# B&R Automation Studio project MotionTestBenchMaster (part 30)

```iecst
                               VAR_RNS_SEQ.Mem.ContainersStop := TRUE;                                                 (* STEP: 51 *)
                               VAR_RNS_SEQ.Mem.ControlInsercion := FALSE;                                              (* STEP: 51 *)
                               VAR_RNS_SEQ.Mem.ControlContinous := FALSE;                                              (* STEP: 51 *)
                               VAR_RNS_SEQ.Mem.PBAbortEnable := FALSE;                                                 (* STEP: 51 PB Abort Sequence Enable*)
                               VAR_RNS_SEQ.Mem.PBStopEnable := TRUE;                                                   (* STEP: 51 PB Stop Sequence Enable*)
                               VAR_RNS_SEQ.Mem.PBStartEnable := FALSE;                                                 (* STEP: 51 PB Start Sequence Enable*)
                               VAR_RNS_SEQ.Mem.ByPassed := FALSE;                                                      (* STEP: 51 *)
                               VAR_RNS_SEQ.Mem.InsercionDevice := FALSE;                                               (* STEP: 51 *)
                               VAR_RNS_SEQ.Mem.AirTreatmentControl := FALSE;                                           (* STEP: 51 *)
                               VAR_RNS_SEQ.Mem.WaterTreatmentControl := FALSE;                                         (* STEP: 51 *)
                               VAR_RNS_SEQ.Mem.SpeedReductionControl := FALSE;                                         (* STEP: 51 *)
                               VAR_RNS_SEQ.Mem.ByPassRequest := FALSE;                                                 (* STEP: 51 *)
                               VAR_RNS_SEQ.Mem.CopAfterCipRequest := FALSE;                                            (* STEP: 51 *)
                               VAR_RNS_SEQ.Mem.NoBoNoSprayInsercion := FALSE;                                          (* STEP: 51 *)

                               VAR_RNS_SEQ.ITC.WTT_ProductRequest := FALSE;                                            (* STEP: 51 *)
                               VAR_RNS_SEQ.ITC.WTT_ProductionRunning := FALSE;                                         (* STEP: 51 *)

                       52..53: (* Spare Steps *)

                       54: (* DRAINING - Stopped *)

                               VAR_RNS_SEQ.Device.AVB224.AutoCnd := TRUE;                                              (* STEP: 54 AVB224*)
                               VAR_RNS_SEQ.Device.AVB224.EnableCnd := FALSE;
                               VAR_RNS_SEQ.Device.AVB228.AutoCnd := FALSE;                                             (* STEP: 54 AVB228*)
                               VAR_RNS_SEQ.Device.AVB228.EnableCnd := FALSE;
                               VAR_RNS_SEQ.Device.AVB234.AutoCnd := TRUE;                                              (* STEP: 54 AVB234*)
                               VAR_RNS_SEQ.Device.AVB234.EnableCnd := FALSE;
                               VAR_RNS_SEQ.Device.AVB261.AutoCnd := FALSE;                                             (* STEP: 54 AVB261*)
                               VAR_RNS_SEQ.Device.AVB261.EnableCnd := FALSE;
                               VAR_RNS_SEQ.Device.AVB264.AutoCnd := FALSE;                                             (* STEP: 54 AVB264*)
                               VAR_RNS_SEQ.Device.AVB264.EnableCnd := FALSE;
                               VAR_RNS_SEQ.Device.AVB265.AutoCnd := FALSE;                                             (* STEP: 54 AVB265*)
                               VAR_RNS_SEQ.Device.AVB265.EnableCnd := FALSE;
                               VAR_RNS_SEQ.Device.AVB266.AutoCnd := TRUE;                                              (* STEP: 54 AVB266*)
                               VAR_RNS_SEQ.Device.AVB266.EnableCnd := FALSE;
                               VAR_RNS_SEQ.Device.AVB267.AutoCnd := TRUE;                                              (* STEP: 54 AVB267*)
                               VAR_RNS_SEQ.Device.AVB267.EnableCnd := FALSE;
                               VAR_RNS_SEQ.Device.AVB268.AutoCnd := TRUE;                                              (* STEP: 54 AVB268*)
                               VAR_RNS_SEQ.Device.AVB268.EnableCnd := FALSE;
                               VAR_RNS_SEQ.Device.AVB273.AutoCnd := FALSE;                                             (* STEP: 54 AVB273*)
                               VAR_RNS_SEQ.Device.AVB273.EnableCnd := FALSE;
                               VAR_RNS_SEQ.Device.AVB294.AutoCnd := FALSE;                                             (* STEP: 54 AVB294*)
                               VAR_RNS_SEQ.Device.AVB294.EnableCnd := FALSE;

                               VAR_RNS_SEQ.Device.PPB209_PID.PID_Enable := FALSE;                                      (* STEP: 54 PPB209*)
                               VAR_RNS_SEQ.Device.PPB209_PID.PID_Mode := FALSE;
                               VAR_RNS_SEQ.Device.PPB209_PID.Auto_SP_Value := 0;
                               VAR_RNS_SEQ.Device.PPB209_PID.FIX_Value := 0;

                               VAR_RNS_SEQ.Device.RVB202_PID.PID_Enable := FALSE;                                      (* STEP: 54 *)
                               VAR_RNS_SEQ.Device.RVB202_PID.PID_Mode := FALSE;
                               VAR_RNS_SEQ.Device.RVB202_PID.Auto_SP_Value := 0;
                               VAR_RNS_SEQ.Device.RVB202_PID.FIX_Value := 0;

                               VAR_RNS_SEQ.Device.FSB220.ALR := FALSE;                                                 (* STEP: 54 FSB220*)
                               VAR_RNS_SEQ.Device.FSB220.WAIT_OFF := FALSE;
                               VAR_RNS_SEQ.Device.FSB220.WAIT_ON := FALSE;

                               VAR_RNS_SEQ.Device.LSB209.ALR := FALSE;                                                 (* STEP: 54 LSB209*)
                               VAR_RNS_SEQ.Device.LSB209.WAIT_OFF := FALSE;
                               VAR_RNS_SEQ.Device.LSB209.WAIT_ON := FALSE;

                               VAR_RNS_SEQ.Device.LSB210.ALR := FALSE;                                                 (* STEP: 54 LSB210*)
                               VAR_RNS_SEQ.Device.LSB210.WAIT_OFF := FALSE;
                               VAR_RNS_SEQ.Device.LSB210.WAIT_ON := FALSE;

                               VAR_RNS_SEQ.Device.LSB299.ALR := FALSE;                                                 (* STEP: 54 *)
                               VAR_RNS_SEQ.Device.LSB299.WAIT_OFF := FALSE;
                               VAR_RNS_SEQ.Device.LSB299.WAIT_ON := FALSE;

                               VAR_RNS_SEQ.Device.FSB201.ALR := FALSE;                                                 (* STEP: 54 FSB201*)
                               VAR_RNS_SEQ.Device.FSB201.WAIT_OFF := FALSE;
                               VAR_RNS_SEQ.Device.FSB201.WAIT_ON := FALSE;

                               VAR_RNS_SEQ.Device.FTB201.ALR_HighLimitEn := FALSE;                                     (* STEP: 54 FTB201*)
                               VAR_RNS_SEQ.Device.FTB201.ALR_HighLimitSP := 0;
                               VAR_RNS_SEQ.Device.FTB201.ALR_LowLimitEn := FALSE;
                               VAR_RNS_SEQ.Device.FTB201.ALR_LowLimitSP := 0;
                               VAR_RNS_SEQ.Device.FTB201.SP := 0;
                               VAR_RNS_SEQ.Device.FTB201.CMP := 0;
                               VAR_RNS_SEQ.Device.FTB201.MinDev := 0;
                               VAR_RNS_SEQ.Device.FTB201.MaxDev := 0;

                               VAR_RNS_SEQ.Device.FTB202.ALR_HighLimitEn := FALSE;                                     (* STEP: 54 FTB202*)
                               VAR_RNS_SEQ.Device.FTB202.ALR_HighLimitSP := 0;
                               VAR_RNS_SEQ.Device.FTB202.ALR_LowLimitEn := FALSE;
                               VAR_RNS_SEQ.Device.FTB202.ALR_LowLimitSP := 0;
                               VAR_RNS_SEQ.Device.FTB202.SP := 0;
                               VAR_RNS_SEQ.Device.FTB202.CMP := 0;
                               VAR_RNS_SEQ.Device.FTB202.MinDev := 0;
                               VAR_RNS_SEQ.Device.FTB202.MaxDev := 0;

                               VAR_RNS_SEQ.Device.PTB220.ALR_HighLimitEn := FALSE;                                     (* STEP: 54 PTB220*)
                               VAR_RNS_SEQ.Device.PTB220.ALR_HighLimitSP := 0;
                               VAR_RNS_SEQ.Device.PTB220.ALR_LowLimitEn := FALSE;
                               VAR_RNS_SEQ.Device.PTB220.ALR_LowLimitSP := 0;
                               VAR_RNS_SEQ.Device.PTB220.SP := 0;
                               VAR_RNS_SEQ.Device.PTB220.CMP := 0;
                               VAR_RNS_SEQ.Device.PTB220.MinDev := 0;
                               VAR_RNS_SEQ.Device.PTB220.MaxDev := 0;

                               VAR_RNS_SEQ.Device.PTB270.ALR_HighLimitEn := FALSE;                                     (* STEP: 54 PTB270*)
                               VAR_RNS_SEQ.Device.PTB270.ALR_HighLimitSP := 0;
                               VAR_RNS_SEQ.Device.PTB270.ALR_LowLimitEn := FALSE;
                               VAR_RNS_SEQ.Device.PTB270.ALR_LowLimitSP := 0;
                               VAR_RNS_SEQ.Device.PTB270.SP := 0;
                               VAR_RNS_SEQ.Device.PTB270.CMP := 0;
                               VAR_RNS_SEQ.Device.PTB270.MinDev := 0;
                               VAR_RNS_SEQ.Device.PTB270.MaxDev := 0;

                               VAR_RNS_SEQ.Device.LTB202.ALR_HighLimitEn := FALSE;                                     (* STEP: 54 LTB202*)
                               VAR_RNS_SEQ.Device.LTB202.ALR_HighLimitSP := 0;
                               VAR_RNS_SEQ.Device.LTB202.ALR_LowLimitEn := FALSE;
                               VAR_RNS_SEQ.Device.LTB202.ALR_LowLimitSP := 0;
                               VAR_RNS_SEQ.Device.LTB202.SP := 0;
                               VAR_RNS_SEQ.Device.LTB202.CMP := 0;
                               VAR_RNS_SEQ.Device.LTB202.MinDev := 0;
                               VAR_RNS_SEQ.Device.LTB202.MaxDev := 0;

                               VAR_RNS_SEQ.Device.PTB290.ALR_HighLimitEn := FALSE;                                     (* STEP: 54 PTB290*)
                               VAR_RNS_SEQ.Device.PTB290.ALR_HighLimitSP := 0;
                               VAR_RNS_SEQ.Device.PTB290.ALR_LowLimitEn := FALSE;
                               VAR_RNS_SEQ.Device.PTB290.ALR_LowLimitSP := 0;
                               VAR_RNS_SEQ.Device.PTB290.SP := 0;
                               VAR_RNS_SEQ.Device.PTB290.CMP := 0;
                               VAR_RNS_SEQ.Device.PTB290.MinDev := 0;
                               VAR_RNS_SEQ.Device.PTB290.MaxDev := 0;

                               VAR_RNS_SEQ.Mem.ContainersStop := TRUE;                                                 (* STEP: 54 *)
                               VAR_RNS_SEQ.Mem.ControlInsercion := FALSE;                                              (* STEP: 54 *)
                               VAR_RNS_SEQ.Mem.ControlContinous := FALSE;                                              (* STEP: 54 *)
                               VAR_RNS_SEQ.Mem.PBAbortEnable := FALSE;                                                 (* STEP: 54 PB Abort Sequence Enable*)
                               VAR_RNS_SEQ.Mem.PBStopEnable := TRUE;                                                   (* STEP: 54 PB Stop Sequence Enable*)
                               VAR_RNS_SEQ.Mem.PBStartEnable := FALSE;                                                 (* STEP: 54 PB Start Sequence Enable*)
                               VAR_RNS_SEQ.Mem.ByPassed := FALSE;                                                      (* STEP: 54 *)
                               VAR_RNS_SEQ.Mem.InsercionDevice := FALSE;                                               (* STEP: 54 *)
                               VAR_RNS_SEQ.Mem.AirTreatmentControl := FALSE;                                           (* STEP: 54 *)
                               VAR_RNS_SEQ.Mem.WaterTreatmentControl := FALSE;                                         (* STEP: 54 *)
                               VAR_RNS_SEQ.Mem.SpeedReductionControl := FALSE;                                         (* STEP: 54 *)
                               VAR_RNS_SEQ.Mem.ByPassRequest := FALSE;                                                 (* STEP: 54 *)
                               VAR_RNS_SEQ.Mem.CopAfterCipRequest := FALSE;                                            (* STEP: 54 *)
                               VAR_RNS_SEQ.Mem.NoBoNoSprayInsercion := FALSE;                                          (* STEP: 54 *)

                               VAR_RNS_SEQ.ITC.WTT_ProductRequest := FALSE;                                            (* STEP: 54 *)
                               VAR_RNS_SEQ.ITC.WTT_ProductionRunning := FALSE;                                         (* STEP: 54 *)

                       55: (* DRAINING - Circuit emptying during COP *)

                               VAR_RNS_SEQ.Device.AVB224.AutoCnd := FALSE;                                             (* STEP: 55 AVB224*)
                               VAR_RNS_SEQ.Device.AVB224.EnableCnd := FALSE;
                               VAR_RNS_SEQ.Device.AVB228.AutoCnd := FALSE;                                             (* STEP: 55 AVB228*)
                               VAR_RNS_SEQ.Device.AVB228.EnableCnd := FALSE;
                               VAR_RNS_SEQ.Device.AVB234.AutoCnd := FALSE;                                             (* STEP: 55 AVB234*)
                               VAR_RNS_SEQ.Device.AVB234.EnableCnd := FALSE;
                               VAR_RNS_SEQ.Device.AVB261.AutoCnd := FALSE;                                             (* STEP: 55 AVB261*)
                               VAR_RNS_SEQ.Device.AVB261.EnableCnd := FALSE;
                               VAR_RNS_SEQ.Device.AVB264.AutoCnd := FALSE;                                             (* STEP: 55 AVB264*)
                               VAR_RNS_SEQ.Device.AVB264.EnableCnd := FALSE;
                               VAR_RNS_SEQ.Device.AVB265.AutoCnd := FALSE;                                             (* STEP: 55 AVB265*)
                               VAR_RNS_SEQ.Device.AVB265.EnableCnd := FALSE;
                               VAR_RNS_SEQ.Device.AVB266.AutoCnd := FALSE;                                             (* STEP: 55 AVB266*)
                               VAR_RNS_SEQ.Device.AVB266.EnableCnd := FALSE;
                               VAR_RNS_SEQ.Device.AVB267.AutoCnd := FALSE;                                             (* STEP: 55 AVB267*)
                               VAR_RNS_SEQ.Device.AVB267.EnableCnd := FALSE;
                               VAR_RNS_SEQ.Device.AVB268.AutoCnd := TRUE;                                              (* STEP: 55 AVB268*)
                               VAR_RNS_SEQ.Device.AVB268.EnableCnd := FALSE;
                               VAR_RNS_SEQ.Device.AVB273.AutoCnd := FALSE;                                             (* STEP: 55 AVB273*)
                               VAR_RNS_SEQ.Device.AVB273.EnableCnd := FALSE;
                               VAR_RNS_SEQ.Device.AVB294.AutoCnd := FALSE;                                             (* STEP: 55 AVB294*)
                               VAR_RNS_SEQ.Device.AVB294.EnableCnd := FALSE;

                               VAR_RNS_SEQ.Device.PPB209_PID.PID_Enable := FALSE;                                      (* STEP: 55 PPB209*)
                               VAR_RNS_SEQ.Device.PPB209_PID.PID_Mode := FALSE;
                               VAR_RNS_SEQ.Device.PPB209_PID.Auto_SP_Value := 0;
                               VAR_RNS_SEQ.Device.PPB209_PID.FIX_Value := 0;

                               VAR_RNS_SEQ.Device.RVB202_PID.PID_Enable := FALSE;                                      (* STEP: 55 *)
                               VAR_RNS_SEQ.Device.RVB202_PID.PID_Mode := FALSE;
                               VAR_RNS_SEQ.Device.RVB202_PID.Auto_SP_Value := 0;
                               VAR_RNS_SEQ.Device.RVB202_PID.FIX_Value := 0;

                               VAR_RNS_SEQ.Device.FSB220.ALR := FALSE;                                                 (* STEP: 55 FSB220*)
                               VAR_RNS_SEQ.Device.FSB220.WAIT_OFF := FALSE;
                               VAR_RNS_SEQ.Device.FSB220.WAIT_ON := FALSE;

                               VAR_RNS_SEQ.Device.LSB209.ALR := FALSE;                                                 (* STEP: 55 LSB209*)
                               VAR_RNS_SEQ.Device.LSB209.WAIT_OFF := FALSE;
                               VAR_RNS_SEQ.Device.LSB209.WAIT_ON := FALSE;

                               VAR_RNS_SEQ.Device.LSB210.ALR := FALSE;                                                 (* STEP: 55 LSB210*)
                               VAR_RNS_SEQ.Device.LSB210.WAIT_OFF := FALSE;
                               VAR_RNS_SEQ.Device.LSB210.WAIT_ON := FALSE;

                               VAR_RNS_SEQ.Device.LSB299.ALR := FALSE;                                                 (* STEP: 55 *)
                               VAR_RNS_SEQ.Device.LSB299.WAIT_OFF := FALSE;
                               VAR_RNS_SEQ.Device.LSB299.WAIT_ON := FALSE;

                               VAR_RNS_SEQ.Device.FSB201.ALR := FALSE;                                                 (* STEP: 55 FSB201*)
                               VAR_RNS_SEQ.Device.FSB201.WAIT_OFF := FALSE;
                               VAR_RNS_SEQ.Device.FSB201.WAIT_ON := FALSE;

                               VAR_RNS_SEQ.Device.FTB201.ALR_HighLimitEn := FALSE;                                     (* STEP: 55 FTB201*)
                               VAR_RNS_SEQ.Device.FTB201.ALR_HighLimitSP := 0;
                               VAR_RNS_SEQ.Device.FTB201.ALR_LowLimitEn := FALSE;
                               VAR_RNS_SEQ.Device.FTB201.ALR_LowLimitSP := 0;
                               VAR_RNS_SEQ.Device.FTB201.SP := 0;
                               VAR_RNS_SEQ.Device.FTB201.CMP := 0;
                               VAR_RNS_SEQ.Device.FTB201.MinDev := 0;
                               VAR_RNS_SEQ.Device.FTB201.MaxDev := 0;

                               VAR_RNS_SEQ.Device.FTB202.ALR_HighLimitEn := FALSE;                                     (* STEP: 55 FTB202*)
                               VAR_RNS_SEQ.Device.FTB202.ALR_HighLimitSP := 0;
                               VAR_RNS_SEQ.Device.FTB202.ALR_LowLimitEn := FALSE;
                               VAR_RNS_SEQ.Device.FTB202.ALR_LowLimitSP := 0;
                               VAR_RNS_SEQ.Device.FTB202.SP := 0;
                               VAR_RNS_SEQ.Device.FTB202.CMP := 0;
                               VAR_RNS_SEQ.Device.FTB202.MinDev := 0;
                               VAR_RNS_SEQ.Device.FTB202.MaxDev := 0;

                               VAR_RNS_SEQ.Device.PTB220.ALR_HighLimitEn := FALSE;                                     (* STEP: 55 PTB220*)
                               VAR_RNS_SEQ.Device.PTB220.ALR_HighLimitSP := 0;
                               VAR_RNS_SEQ.Device.PTB220.ALR_LowLimitEn := FALSE;
                               VAR_RNS_SEQ.Device.PTB220.ALR_LowLimitSP := 0;
                               VAR_RNS_SEQ.Device.PTB220.SP := 0;
                               VAR_RNS_SEQ.Device.PTB220.CMP := 0;
                               VAR_RNS_SEQ.Device.PTB220.MinDev := 0;
                               VAR_RNS_SEQ.Device.PTB220.MaxDev := 0;

                               VAR_RNS_SEQ.Device.PTB270.ALR_HighLimitEn := FALSE;                                     (* STEP: 55 PTB270*)
                               VAR_RNS_SEQ.Device.PTB270.ALR_HighLimitSP := 0;
                               VAR_RNS_SEQ.Device.PTB270.ALR_LowLimitEn := FALSE;
                               VAR_RNS_SEQ.Device.PTB270.ALR_LowLimitSP := 0;
                               VAR_RNS_SEQ.Device.PTB270.SP := 0;
                               VAR_RNS_SEQ.Device.PTB270.CMP := 0;
                               VAR_RNS_SEQ.Device.PTB270.MinDev := 0;
                               VAR_RNS_SEQ.Device.PTB270.MaxDev := 0;

                               VAR_RNS_SEQ.Device.LTB202.ALR_HighLimitEn := FALSE;                                     (* STEP: 55 LTB202*)
                               VAR_RNS_SEQ.Device.LTB202.ALR_HighLimitSP := 0;
                               VAR_RNS_SEQ.Device.LTB202.ALR_LowLimitEn := FALSE;
                               VAR_RNS_SEQ.Device.LTB202.ALR_LowLimitSP := 0;
                               VAR_RNS_SEQ.Device.LTB202.SP := 0;
                               VAR_RNS_SEQ.Device.LTB202.CMP := 0;
                               VAR_RNS_SEQ.Device.LTB202.MinDev := 0;
                               VAR_RNS_SEQ.Device.LTB202.MaxDev := 0;

                               VAR_RNS_SEQ.Device.PTB290.ALR_HighLimitEn := FALSE;                                     (* STEP: 55 PTB290*)
                               VAR_RNS_SEQ.Device.PTB290.ALR_HighLimitSP := 0;
                               VAR_RNS_SEQ.Device.PTB290.ALR_LowLimitEn := FALSE;
                               VAR_RNS_SEQ.Device.PTB290.ALR_LowLimitSP := 0;
                               VAR_RNS_SEQ.Device.PTB290.SP := 0;
                               VAR_RNS_SEQ.Device.PTB290.CMP := 0;
                               VAR_RNS_SEQ.Device.PTB290.MinDev := 0;
                               VAR_RNS_SEQ.Device.PTB290.MaxDev := 0;

                               VAR_RNS_SEQ.Mem.ContainersStop := TRUE;                                                 (* STEP: 55 *)
                               VAR_RNS_SEQ.Mem.ControlInsercion := FALSE;                                              (* STEP: 55 *)
                               VAR_RNS_SEQ.Mem.ControlContinous := FALSE;                                              (* STEP: 55 *)
                               VAR_RNS_SEQ.Mem.PBAbortEnable := FALSE;                                                 (* STEP: 55 PB Abort Sequence Enable*)
                               VAR_RNS_SEQ.Mem.PBStopEnable := FALSE;                                                  (* STEP: 55 PB Stop Sequence Enable*)
                               VAR_RNS_SEQ.Mem.PBStartEnable := FALSE;                                                 (* STEP: 55 PB Start Sequence Enable*)
                               VAR_RNS_SEQ.Mem.ByPassed := FALSE;                                                      (* STEP: 55 *)
                               VAR_RNS_SEQ.Mem.InsercionDevice := FALSE;                                               (* STEP: 55 *)
                               VAR_RNS_SEQ.Mem.AirTreatmentControl := FALSE;                                           (* STEP: 55 *)
                               VAR_RNS_SEQ.Mem.WaterTreatmentControl := FALSE;                                         (* STEP: 55 *)
                               VAR_RNS_SEQ.Mem.SpeedReductionControl := TRUE;                                          (* STEP: 55 *)
                               VAR_RNS_SEQ.Mem.ByPassRequest := FALSE;                                                 (* STEP: 55 *)
                               VAR_RNS_SEQ.Mem.CopAfterCipRequest := TRUE;                                             (* STEP: 55 *)
                               VAR_RNS_SEQ.Mem.NoBoNoSprayInsercion := FALSE;                                          (* STEP: 55 *)

                               VAR_RNS_SEQ.ITC.WTT_ProductRequest := FALSE;                                            (* STEP: 55 *)
                               VAR_RNS_SEQ.ITC.WTT_ProductionRunning := FALSE;                                         (* STEP: 55 *)

                       56..69: (* Spare Steps *)

                       70: (* CONTROL - Check Selection and Speed *)

                               VAR_RNS_SEQ.Device.AVB224.AutoCnd := FALSE;                                             (* STEP: 70 AVB224*)
                               VAR_RNS_SEQ.Device.AVB224.EnableCnd := FALSE;
                               VAR_RNS_SEQ.Device.AVB228.AutoCnd := FALSE;                                             (* STEP: 70 AVB228*)
                               VAR_RNS_SEQ.Device.AVB228.EnableCnd := FALSE;
                               VAR_RNS_SEQ.Device.AVB234.AutoCnd := FALSE;                                             (* STEP: 70 AVB234*)
                               VAR_RNS_SEQ.Device.AVB234.EnableCnd := FALSE;
                               VAR_RNS_SEQ.Device.AVB261.AutoCnd := FALSE;                                             (* STEP: 70 AVB261*)
                               VAR_RNS_SEQ.Device.AVB261.EnableCnd := FALSE;
                               VAR_RNS_SEQ.Device.AVB264.AutoCnd := FALSE;                                             (* STEP: 70 AVB264*)
                               VAR_RNS_SEQ.Device.AVB264.EnableCnd := FALSE;
                               VAR_RNS_SEQ.Device.AVB265.AutoCnd := FALSE;                                             (* STEP: 70 AVB265*)
                               VAR_RNS_SEQ.Device.AVB265.EnableCnd := FALSE;
                               VAR_RNS_SEQ.Device.AVB266.AutoCnd := FALSE;                                             (* STEP: 70 AVB266*)
                               VAR_RNS_SEQ.Device.AVB266.EnableCnd := FALSE;
                               VAR_RNS_SEQ.Device.AVB267.AutoCnd := FALSE;                                             (* STEP: 70 AVB267*)
                               VAR_RNS_SEQ.Device.AVB267.EnableCnd := FALSE;
                               VAR_RNS_SEQ.Device.AVB268.AutoCnd := FALSE;                                             (* STEP: 70 AVB268*)
                               VAR_RNS_SEQ.Device.AVB268.EnableCnd := FALSE;
                               VAR_RNS_SEQ.Device.AVB273.AutoCnd := FALSE;                                             (* STEP: 70 AVB273*)
                               VAR_RNS_SEQ.Device.AVB273.EnableCnd := FALSE;
                               VAR_RNS_SEQ.Device.AVB294.AutoCnd := FALSE;                                             (* STEP: 70 AVB294*)
                               VAR_RNS_SEQ.Device.AVB294.EnableCnd := FALSE;

                               VAR_RNS_SEQ.Device.PPB209_PID.PID_Enable := FALSE;                                      (* STEP: 70 PPB209*)
                               VAR_RNS_SEQ.Device.PPB209_PID.PID_Mode := FALSE;
                               VAR_RNS_SEQ.Device.PPB209_PID.Auto_SP_Value := 0;
                               VAR_RNS_SEQ.Device.PPB209_PID.FIX_Value := 0;

                               VAR_RNS_SEQ.Device.RVB202_PID.PID_Enable := FALSE;                                      (* STEP: 70 *)
                               VAR_RNS_SEQ.Device.RVB202_PID.PID_Mode := FALSE;
                               VAR_RNS_SEQ.Device.RVB202_PID.Auto_SP_Value := 0;
                               VAR_RNS_SEQ.Device.RVB202_PID.FIX_Value := 0;

                               VAR_RNS_SEQ.Device.FSB220.ALR := FALSE;                                                 (* STEP: 70 FSB220*)
                               VAR_RNS_SEQ.Device.FSB220.WAIT_OFF := FALSE;
                               VAR_RNS_SEQ.Device.FSB220.WAIT_ON := FALSE;

                               VAR_RNS_SEQ.Device.LSB209.ALR := FALSE;                                                 (* STEP: 70 LSB209*)
                               VAR_RNS_SEQ.Device.LSB209.WAIT_OFF := FALSE;
                               VAR_RNS_SEQ.Device.LSB209.WAIT_ON := FALSE;

                               VAR_RNS_SEQ.Device.LSB210.ALR := FALSE;                                                 (* STEP: 70 LSB210*)
                               VAR_RNS_SEQ.Device.LSB210.WAIT_OFF := FALSE;
                               VAR_RNS_SEQ.Device.LSB210.WAIT_ON := FALSE;

                               VAR_RNS_SEQ.Device.LSB299.ALR := FALSE;                                                 (* STEP: 70 *)
                               VAR_RNS_SEQ.Device.LSB299.WAIT_OFF := FALSE;
                               VAR_RNS_SEQ.Device.LSB299.WAIT_ON := FALSE;

                               VAR_RNS_SEQ.Device.FSB201.ALR := FALSE;                                                 (* STEP: 70 FSB201*)
                               VAR_RNS_SEQ.Device.FSB201.WAIT_OFF := FALSE;
                               VAR_RNS_SEQ.Device.FSB201.WAIT_ON := FALSE;

                               VAR_RNS_SEQ.Device.FTB201.ALR_HighLimitEn := FALSE;                                     (* STEP: 70 FTB201*)
                               VAR_RNS_SEQ.Device.FTB201.ALR_HighLimitSP := 0;
                               VAR_RNS_SEQ.Device.FTB201.ALR_LowLimitEn := FALSE;
                               VAR_RNS_SEQ.Device.FTB201.ALR_LowLimitSP := 0;
                               VAR_RNS_SEQ.Device.FTB201.SP := 0;
                               VAR_RNS_SEQ.Device.FTB201.CMP := 0;
                               VAR_RNS_SEQ.Device.FTB201.MinDev := 0;
                               VAR_RNS_SEQ.Device.FTB201.MaxDev := 0;

                               VAR_RNS_SEQ.Device.FTB202.ALR_HighLimitEn := FALSE;                                     (* STEP: 70 FTB202*)
                               VAR_RNS_SEQ.Device.FTB202.ALR_HighLimitSP := 0;
                               VAR_RNS_SEQ.Device.FTB202.ALR_LowLimitEn := FALSE;
                               VAR_RNS_SEQ.Device.FTB202.ALR_LowLimitSP := 0;
                               VAR_RNS_SEQ.Device.FTB202.SP := 0;
                               VAR_RNS_SEQ.Device.FTB202.CMP := 0;
                               VAR_RNS_SEQ.Device.FTB202.MinDev := 0;
                               VAR_RNS_SEQ.Device.FTB202.MaxDev := 0;

                               VAR_RNS_SEQ.Device.PTB220.ALR_HighLimitEn := FALSE;                                     (* STEP: 70 PTB220*)
                               VAR_RNS_SEQ.Device.PTB220.ALR_HighLimitSP := 0;
                               VAR_RNS_SEQ.Device.PTB220.ALR_LowLimitEn := FALSE;
                               VAR_RNS_SEQ.Device.PTB220.ALR_LowLimitSP := 0;
                               VAR_RNS_SEQ.Device.PTB220.SP := 0;
                               VAR_RNS_SEQ.Device.PTB220.CMP := 0;
                               VAR_RNS_SEQ.Device.PTB220.MinDev := 0;
                               VAR_RNS_SEQ.Device.PTB220.MaxDev := 0;

                               VAR_RNS_SEQ.Device.PTB270.ALR_HighLimitEn := FALSE;                                     (* STEP: 70 PTB270*)
                               VAR_RNS_SEQ.Device.PTB270.ALR_HighLimitSP := 0;
                               VAR_RNS_SEQ.Device.PTB270.ALR_LowLimitEn := FALSE;
                               VAR_RNS_SEQ.Device.PTB270.ALR_LowLimitSP := 0;
                               VAR_RNS_SEQ.Device.PTB270.SP := 0;
                               VAR_RNS_SEQ.Device.PTB270.CMP := 0;
                               VAR_RNS_SEQ.Device.PTB270.MinDev := 0;
                               VAR_RNS_SEQ.Device.PTB270.MaxDev := 0;

                               VAR_RNS_SEQ.Device.LTB202.ALR_HighLimitEn := FALSE;                                     (* STEP: 70 LTB202*)
                               VAR_RNS_SEQ.Device.LTB202.ALR_HighLimitSP := 0;
                               VAR_RNS_SEQ.Device.LTB202.ALR_LowLimitEn := FALSE;
                               VAR_RNS_SEQ.Device.LTB202.ALR_LowLimitSP := 0;
                               VAR_RNS_SEQ.Device.LTB202.SP := 0;
                               VAR_RNS_SEQ.Device.LTB202.CMP := 0;
                               VAR_RNS_SEQ.Device.LTB202.MinDev := 0;
                               VAR_RNS_SEQ.Device.LTB202.MaxDev := 0;

                               VAR_RNS_SEQ.Device.PTB290.ALR_HighLimitEn := FALSE;                                     (* STEP: 70 PTB290*)
                               VAR_RNS_SEQ.Device.PTB290.ALR_HighLimitSP := 0;
                               VAR_RNS_SEQ.Device.PTB290.ALR_LowLimitEn := FALSE;
                               VAR_RNS_SEQ.Device.PTB290.ALR_LowLimitSP := 0;
                               VAR_RNS_SEQ.Device.PTB290.SP := 0;
                               VAR_RNS_SEQ.Device.PTB290.CMP := 0;
                               VAR_RNS_SEQ.Device.PTB290.MinDev := 0;
                               VAR_RNS_SEQ.Device.PTB290.MaxDev := 0;

                               VAR_RNS_SEQ.Mem.ContainersStop := TRUE;                                                 (* STEP: 70 *)
                               VAR_RNS_SEQ.Mem.ControlInsercion := FALSE;                                              (* STEP: 70 *)
                               VAR_RNS_SEQ.Mem.ControlContinous := FALSE;                                              (* STEP: 70 *)
                               VAR_RNS_SEQ.Mem.PBAbortEnable := TRUE;                                                  (* STEP: 70 PB Abort Sequence Enable*)
                               VAR_RNS_SEQ.Mem.PBStopEnable := TRUE;                                                   (* STEP: 70 PB Stop Sequence Enable*)
                               VAR_RNS_SEQ.Mem.PBStartEnable := FALSE;                                                 (* STEP: 70 PB Start Sequence Enable*)
                               VAR_RNS_SEQ.Mem.ByPassed := FALSE;                                                      (* STEP: 70 *)
                               VAR_RNS_SEQ.Mem.InsercionDevice := FALSE;                                               (* STEP: 70 *)
                               VAR_RNS_SEQ.Mem.AirTreatmentControl := FALSE;                                           (* STEP: 70 *)
                               VAR_RNS_SEQ.Mem.WaterTreatmentControl := FALSE;                                         (* STEP: 70 *)
                               VAR_RNS_SEQ.Mem.SpeedReductionControl := TRUE;                                          (* STEP: 70 *)
                               VAR_RNS_SEQ.Mem.ByPassRequest := FALSE;                                                 (* STEP: 70 *)
                               VAR_RNS_SEQ.Mem.CopAfterCipRequest := FALSE;                                            (* STEP: 70 *)
                               VAR_RNS_SEQ.Mem.NoBoNoSprayInsercion := FALSE;                                          (* STEP: 70 *)

                               VAR_RNS_SEQ.ITC.WTT_ProductRequest := FALSE;                                            (* STEP: 70 *)
                               VAR_RNS_SEQ.ITC.WTT_ProductionRunning := FALSE;                                         (* STEP: 70 *)

                       71: (* CONTROL - Insercion Device *)

                               VAR_RNS_SEQ.Device.AVB224.AutoCnd := FALSE;                                             (* STEP: 71 AVB224*)
                               VAR_RNS_SEQ.Device.AVB224.EnableCnd := FALSE;
                               VAR_RNS_SEQ.Device.AVB228.AutoCnd := TRUE;                                              (* STEP: 71 AVB228*)
                               VAR_RNS_SEQ.Device.AVB228.EnableCnd := FALSE;
                               VAR_RNS_SEQ.Device.AVB234.AutoCnd := FALSE;                                             (* STEP: 71 AVB234*)
                               VAR_RNS_SEQ.Device.AVB234.EnableCnd := FALSE;
                               VAR_RNS_SEQ.Device.AVB261.AutoCnd := TRUE;                                              (* STEP: 71 AVB261*)
                               VAR_RNS_SEQ.Device.AVB261.EnableCnd := FALSE;
                               VAR_RNS_SEQ.Device.AVB264.AutoCnd := FALSE;                                             (* STEP: 71 AVB264*)
                               VAR_RNS_SEQ.Device.AVB264.EnableCnd := FALSE;
                               VAR_RNS_SEQ.Device.AVB265.AutoCnd := FALSE;                                             (* STEP: 71 AVB265*)
                               VAR_RNS_SEQ.Device.AVB265.EnableCnd := FALSE;
                               VAR_RNS_SEQ.Device.AVB266.AutoCnd := FALSE;                                             (* STEP: 71 AVB266*)
                               VAR_RNS_SEQ.Device.AVB266.EnableCnd := FALSE;
                               VAR_RNS_SEQ.Device.AVB267.AutoCnd := FALSE;                                             (* STEP: 71 AVB267*)
                               VAR_RNS_SEQ.Device.AVB267.EnableCnd := FALSE;
                               VAR_RNS_SEQ.Device.AVB268.AutoCnd := FALSE;                                             (* STEP: 71 AVB268*)
                               VAR_RNS_SEQ.Device.AVB268.EnableCnd := FALSE;
                               VAR_RNS_SEQ.Device.AVB273.AutoCnd := FALSE;                                             (* STEP: 71 AVB273*)
                               VAR_RNS_SEQ.Device.AVB273.EnableCnd := FALSE;
                               VAR_RNS_SEQ.Device.AVB294.AutoCnd := FALSE;                                             (* STEP: 71 AVB294*)
                               VAR_RNS_SEQ.Device.AVB294.EnableCnd := FALSE;

                               VAR_RNS_SEQ.Device.PPB209_PID.PID_Enable := FALSE;                                      (* STEP: 71 PPB209*)
                               VAR_RNS_SEQ.Device.PPB209_PID.PID_Mode := FALSE;
                               VAR_RNS_SEQ.Device.PPB209_PID.Auto_SP_Value := 0;
                               VAR_RNS_SEQ.Device.PPB209_PID.FIX_Value := 0;

                               VAR_RNS_SEQ.Device.RVB202_PID.PID_Enable := FALSE;                                      (* STEP: 71 *)
                               VAR_RNS_SEQ.Device.RVB202_PID.PID_Mode := FALSE;
                               VAR_RNS_SEQ.Device.RVB202_PID.Auto_SP_Value := 0;
                               VAR_RNS_SEQ.Device.RVB202_PID.FIX_Value := 0;

                               VAR_RNS_SEQ.Device.FSB220.ALR := TRUE;                                                  (* STEP: 71 FSB220*)
                               VAR_RNS_SEQ.Device.FSB220.WAIT_OFF := FALSE;
                               VAR_RNS_SEQ.Device.FSB220.WAIT_ON := TRUE;

                               VAR_RNS_SEQ.Device.LSB209.ALR := FALSE;                                                 (* STEP: 71 LSB209*)
                               VAR_RNS_SEQ.Device.LSB209.WAIT_OFF := FALSE;
                               VAR_RNS_SEQ.Device.LSB209.WAIT_ON := FALSE;

                               VAR_RNS_SEQ.Device.LSB210.ALR := FALSE;                                                 (* STEP: 71 LSB210*)
                               VAR_RNS_SEQ.Device.LSB210.WAIT_OFF := FALSE;
                               VAR_RNS_SEQ.Device.LSB210.WAIT_ON := FALSE;

                               VAR_RNS_SEQ.Device.LSB299.ALR := FALSE;                                                 (* STEP: 71 *)
                               VAR_RNS_SEQ.Device.LSB299.WAIT_OFF := FALSE;
                               VAR_RNS_SEQ.Device.LSB299.WAIT_ON := FALSE;

                               VAR_RNS_SEQ.Device.FSB201.ALR := TRUE;                                                  (* STEP: 71 FSB201*)
                               VAR_RNS_SEQ.Device.FSB201.WAIT_OFF := FALSE;
                               VAR_RNS_SEQ.Device.FSB201.WAIT_ON := TRUE;

                               VAR_RNS_SEQ.Device.FTB201.ALR_HighLimitEn := FALSE;                                     (* STEP: 71 FTB201*)
                               VAR_RNS_SEQ.Device.FTB201.ALR_HighLimitSP := 0;
                               VAR_RNS_SEQ.Device.FTB201.ALR_LowLimitEn := FALSE;
                               VAR_RNS_SEQ.Device.FTB201.ALR_LowLimitSP := 0;
                               VAR_RNS_SEQ.Device.FTB201.SP := 0;
                               VAR_RNS_SEQ.Device.FTB201.CMP := 0;
                               VAR_RNS_SEQ.Device.FTB201.MinDev := 0;
                               VAR_RNS_SEQ.Device.FTB201.MaxDev := 0;

                               VAR_RNS_SEQ.Device.FTB202.ALR_HighLimitEn := FALSE;                                     (* STEP: 71 FTB202*)
                               VAR_RNS_SEQ.Device.FTB202.ALR_HighLimitSP := 0;
                               VAR_RNS_SEQ.Device.FTB202.ALR_LowLimitEn := FALSE;
                               VAR_RNS_SEQ.Device.FTB202.ALR_LowLimitSP := 0;
                               VAR_RNS_SEQ.Device.FTB202.SP := 0;
                               VAR_RNS_SEQ.Device.FTB202.CMP := 0;
                               VAR_RNS_SEQ.Device.FTB202.MinDev := 0;
                               VAR_RNS_SEQ.Device.FTB202.MaxDev := 0;

                               VAR_RNS_SEQ.Device.PTB220.ALR_HighLimitEn := FALSE;                                     (* STEP: 71 PTB220*)
                               VAR_RNS_SEQ.Device.PTB220.ALR_HighLimitSP := 0;
                               VAR_RNS_SEQ.Device.PTB220.ALR_LowLimitEn := FALSE;
                               VAR_RNS_SEQ.Device.PTB220.ALR_LowLimitSP := 0;
                               VAR_RNS_SEQ.Device.PTB220.SP := 0;
                               VAR_RNS_SEQ.Device.PTB220.CMP := 0;
                               VAR_RNS_SEQ.Device.PTB220.MinDev := 0;
                               VAR_RNS_SEQ.Device.PTB220.MaxDev := 0;

                               VAR_RNS_SEQ.Device.PTB270.ALR_HighLimitEn := FALSE;                                     (* STEP: 71 PTB270*)
                               VAR_RNS_SEQ.Device.PTB270.ALR_HighLimitSP := 0;
                               VAR_RNS_SEQ.Device.PTB270.ALR_LowLimitEn := FALSE;
                               VAR_RNS_SEQ.Device.PTB270.ALR_LowLimitSP := 0;
                               VAR_RNS_SEQ.Device.PTB270.SP := 0;
                               VAR_RNS_SEQ.Device.PTB270.CMP := 0;
                               VAR_RNS_SEQ.Device.PTB270.MinDev := 0;
                               VAR_RNS_SEQ.Device.PTB270.MaxDev := 0;

                               VAR_RNS_SEQ.Device.LTB202.ALR_HighLimitEn := FALSE;                                     (* STEP: 71 LTB202*)
                               VAR_RNS_SEQ.Device.LTB202.ALR_HighLimitSP := 0;
                               VAR_RNS_SEQ.Device.LTB202.ALR_LowLimitEn := FALSE;
                               VAR_RNS_SEQ.Device.LTB202.ALR_LowLimitSP := 0;
                               VAR_RNS_SEQ.Device.LTB202.SP := 0;
                               VAR_RNS_SEQ.Device.LTB202.CMP := 0;
                               VAR_RNS_SEQ.Device.LTB202.MinDev := 0;
                               VAR_RNS_SEQ.Device.LTB202.MaxDev := 0;

                               VAR_RNS_SEQ.Device.PTB290.ALR_HighLimitEn := FALSE;                                     (* STEP: 71 PTB290*)
                               VAR_RNS_SEQ.Device.PTB290.ALR_HighLimitSP := 0;
                               VAR_RNS_SEQ.Device.PTB290.ALR_LowLimitEn := FALSE;
                               VAR_RNS_SEQ.Device.PTB290.ALR_LowLimitSP := 0;
                               VAR_RNS_SEQ.Device.PTB290.SP := 0;
                               VAR_RNS_SEQ.Device.PTB290.CMP := 0;
                               VAR_RNS_SEQ.Device.PTB290.MinDev := 0;
                               VAR_RNS_SEQ.Device.PTB290.MaxDev := 0;

                               VAR_RNS_SEQ.Mem.ContainersStop := TRUE;                                                 (* STEP: 71 *)
                               VAR_RNS_SEQ.Mem.ControlInsercion := FALSE;                                              (* STEP: 71 *)
                               VAR_RNS_SEQ.Mem.ControlContinous := FALSE;                                              (* STEP: 71 *)
                               VAR_RNS_SEQ.Mem.PBAbortEnable := TRUE;                                                  (* STEP: 71 PB Abort Sequence Enable*)
                               VAR_RNS_SEQ.Mem.PBStopEnable := TRUE;                                                   (* STEP: 71 PB Stop Sequence Enable*)
                               VAR_RNS_SEQ.Mem.PBStartEnable := FALSE;                                                 (* STEP: 71 PB Start Sequence Enable*)
                               VAR_RNS_SEQ.Mem.ByPassed := FALSE;                                                      (* STEP: 71 *)
                               VAR_RNS_SEQ.Mem.InsercionDevice := TRUE;                                                (* STEP: 71 *)
                               VAR_RNS_SEQ.Mem.AirTreatmentControl := FALSE;                                           (* STEP: 71 *)
                               VAR_RNS_SEQ.Mem.WaterTreatmentControl := FALSE;                                         (* STEP: 71 *)
                               VAR_RNS_SEQ.Mem.SpeedReductionControl := TRUE;                                          (* STEP: 71 *)
                               VAR_RNS_SEQ.Mem.ByPassRequest := FALSE;                                                 (* STEP: 71 *)
                               VAR_RNS_SEQ.Mem.CopAfterCipRequest := FALSE;                                            (* STEP: 71 *)
                               VAR_RNS_SEQ.Mem.NoBoNoSprayInsercion := FALSE;                                          (* STEP: 71 *)

                               VAR_RNS_SEQ.ITC.WTT_ProductRequest := FALSE;                                            (* STEP: 71 *)
                               VAR_RNS_SEQ.ITC.WTT_ProductionRunning := FALSE;                                         (* STEP: 71 *)

                       72: (* CONTROL - Air Startup I *)

                               VAR_RNS_SEQ.Device.AVB224.AutoCnd := FALSE;                                             (* STEP: 72 AVB224*)
                               VAR_RNS_SEQ.Device.AVB224.EnableCnd := FALSE;
                               VAR_RNS_SEQ.Device.AVB228.AutoCnd := FALSE;                                             (* STEP: 72 AVB228*)
                               VAR_RNS_SEQ.Device.AVB228.EnableCnd := FALSE;
                               VAR_RNS_SEQ.Device.AVB234.AutoCnd := FALSE;                                             (* STEP: 72 AVB234*)
                               VAR_RNS_SEQ.Device.AVB234.EnableCnd := FALSE;
                               VAR_RNS_SEQ.Device.AVB261.AutoCnd := FALSE;                                             (* STEP: 72 AVB261*)
                               VAR_RNS_SEQ.Device.AVB261.EnableCnd := FALSE;
                               VAR_RNS_SEQ.Device.AVB264.AutoCnd := FALSE;                                             (* STEP: 72 AVB264*)
                               VAR_RNS_SEQ.Device.AVB264.EnableCnd := FALSE;
                               VAR_RNS_SEQ.Device.AVB265.AutoCnd := FALSE;                                             (* STEP: 72 AVB265*)
                               VAR_RNS_SEQ.Device.AVB265.EnableCnd := FALSE;
                               VAR_RNS_SEQ.Device.AVB266.AutoCnd := FALSE;                                             (* STEP: 72 AVB266*)
                               VAR_RNS_SEQ.Device.AVB266.EnableCnd := FALSE;
                               VAR_RNS_SEQ.Device.AVB267.AutoCnd := FALSE;                                             (* STEP: 72 AVB267*)
                               VAR_RNS_SEQ.Device.AVB267.EnableCnd := FALSE;
                               VAR_RNS_SEQ.Device.AVB268.AutoCnd := FALSE;                                             (* STEP: 72 AVB268*)
                               VAR_RNS_SEQ.Device.AVB268.EnableCnd := FALSE;
                               VAR_RNS_SEQ.Device.AVB273.AutoCnd := TRUE;                                              (* STEP: 72 AVB273*)
                               VAR_RNS_SEQ.Device.AVB273.EnableCnd := FALSE;
                               VAR_RNS_SEQ.Device.AVB294.AutoCnd := FALSE;                                             (* STEP: 72 AVB294*)
                               VAR_RNS_SEQ.Device.AVB294.EnableCnd := FALSE;

                               VAR_RNS_SEQ.Device.PPB209_PID.PID_Enable := FALSE;                                      (* STEP: 72 PPB209*)
                               VAR_RNS_SEQ.Device.PPB209_PID.PID_Mode := FALSE;
                               VAR_RNS_SEQ.Device.PPB209_PID.Auto_SP_Value := 0;
                               VAR_RNS_SEQ.Device.PPB209_PID.FIX_Value := 0;

                               VAR_RNS_SEQ.Device.RVB202_PID.PID_Enable := FALSE;                                      (* STEP: 72 *)
                               VAR_RNS_SEQ.Device.RVB202_PID.PID_Mode := FALSE;
                               VAR_RNS_SEQ.Device.RVB202_PID.Auto_SP_Value := 0;
                               VAR_RNS_SEQ.Device.RVB202_PID.FIX_Value := 0;

                               VAR_RNS_SEQ.Device.FSB220.ALR := FALSE;                                                 (* STEP: 72 FSB220*)
                               VAR_RNS_SEQ.Device.FSB220.WAIT_OFF := FALSE;
                               VAR_RNS_SEQ.Device.FSB220.WAIT_ON := FALSE;

                               VAR_RNS_SEQ.Device.LSB209.ALR := FALSE;                                                 (* STEP: 72 LSB209*)
                               VAR_RNS_SEQ.Device.LSB209.WAIT_OFF := FALSE;
                               VAR_RNS_SEQ.Device.LSB209.WAIT_ON := FALSE;

                               VAR_RNS_SEQ.Device.LSB210.ALR := FALSE;                                                 (* STEP: 72 LSB210*)
                               VAR_RNS_SEQ.Device.LSB210.WAIT_OFF := FALSE;
                               VAR_RNS_SEQ.Device.LSB210.WAIT_ON := FALSE;

                               VAR_RNS_SEQ.Device.LSB299.ALR := FALSE;                                                 (* STEP: 72 *)
                               VAR_RNS_SEQ.Device.LSB299.WAIT_OFF := FALSE;
                               VAR_RNS_SEQ.Device.LSB299.WAIT_ON := FALSE;

                               VAR_RNS_SEQ.Device.FSB201.ALR := FALSE;                                                 (* STEP: 72 FSB201*)
                               VAR_RNS_SEQ.Device.FSB201.WAIT_OFF := FALSE;
                               VAR_RNS_SEQ.Device.FSB201.WAIT_ON := FALSE;

                               VAR_RNS_SEQ.Device.FTB201.ALR_HighLimitEn := FALSE;                                     (* STEP: 72 FTB201*)
                               VAR_RNS_SEQ.Device.FTB201.ALR_HighLimitSP := 0;
                               VAR_RNS_SEQ.Device.FTB201.ALR_LowLimitEn := TRUE;
                               VAR_RNS_SEQ.Device.FTB201.ALR_LowLimitSP := HMI_PAR_1._166;
                               VAR_RNS_SEQ.Device.FTB201.SP := HMI_PAR_1._164;
                               VAR_RNS_SEQ.Device.FTB201.CMP := 3;
                               VAR_RNS_SEQ.Device.FTB201.MinDev := HMI_PAR_1._165;
                               VAR_RNS_SEQ.Device.FTB201.MaxDev := 2*HMI_PAR_1._165;

                               VAR_RNS_SEQ.Device.FTB202.ALR_HighLimitEn := FALSE;                                     (* STEP: 72 FTB202*)
                               VAR_RNS_SEQ.Device.FTB202.ALR_HighLimitSP := 0;
                               VAR_RNS_SEQ.Device.FTB202.ALR_LowLimitEn := FALSE;
                               VAR_RNS_SEQ.Device.FTB202.ALR_LowLimitSP := 0;
                               VAR_RNS_SEQ.Device.FTB202.SP := 0;
                               VAR_RNS_SEQ.Device.FTB202.CMP := 0;
                               VAR_RNS_SEQ.Device.FTB202.MinDev := 0;
                               VAR_RNS_SEQ.Device.FTB202.MaxDev := 0;

                               VAR_RNS_SEQ.Device.PTB220.ALR_HighLimitEn := FALSE;                                     (* STEP: 72 PTB220*)
                               VAR_RNS_SEQ.Device.PTB220.ALR_HighLimitSP := 0;
                               VAR_RNS_SEQ.Device.PTB220.ALR_LowLimitEn := FALSE;
                               VAR_RNS_SEQ.Device.PTB220.ALR_LowLimitSP := 0;
                               VAR_RNS_SEQ.Device.PTB220.SP := 0;
                               VAR_RNS_SEQ.Device.PTB220.CMP := 0;
                               VAR_RNS_SEQ.Device.PTB220.MinDev := 0;
                               VAR_RNS_SEQ.Device.PTB220.MaxDev := 0;

                               VAR_RNS_SEQ.Device.PTB270.ALR_HighLimitEn := FALSE;                                     (* STEP: 72 PTB270*)
                               VAR_RNS_SEQ.Device.PTB270.ALR_HighLimitSP := 0;
                               VAR_RNS_SEQ.Device.PTB270.ALR_LowLimitEn := FALSE;
                               VAR_RNS_SEQ.Device.PTB270.ALR_LowLimitSP := 0;
                               VAR_RNS_SEQ.Device.PTB270.SP := 0;
                               VAR_RNS_SEQ.Device.PTB270.CMP := 0;
                               VAR_RNS_SEQ.Device.PTB270.MinDev := 0;
                               VAR_RNS_SEQ.Device.PTB270.MaxDev := 0;

                               VAR_RNS_SEQ.Device.LTB202.ALR_HighLimitEn := FALSE;                                     (* STEP: 72 LTB202*)
                               VAR_RNS_SEQ.Device.LTB202.ALR_HighLimitSP := 0;
                               VAR_RNS_SEQ.Device.LTB202.ALR_LowLimitEn := FALSE;
                               VAR_RNS_SEQ.Device.LTB202.ALR_LowLimitSP := 0;
                               VAR_RNS_SEQ.Device.LTB202.SP := 0;
                               VAR_RNS_SEQ.Device.LTB202.CMP := 0;
                               VAR_RNS_SEQ.Device.LTB202.MinDev := 0;
                               VAR_RNS_SEQ.Device.LTB202.MaxDev := 0;

                               VAR_RNS_SEQ.Device.PTB290.ALR_HighLimitEn := FALSE;                                     (* STEP: 72 PTB290*)
                               VAR_RNS_SEQ.Device.PTB290.ALR_HighLimitSP := 0;
                               VAR_RNS_SEQ.Device.PTB290.ALR_LowLimitEn := FALSE;
                               VAR_RNS_SEQ.Device.PTB290.ALR_LowLimitSP := 0;
                               VAR_RNS_SEQ.Device.PTB290.SP := 0;
                               VAR_RNS_SEQ.Device.PTB290.CMP := 0;
                               VAR_RNS_SEQ.Device.PTB290.MinDev := 0;
                               VAR_RNS_SEQ.Device.PTB290.MaxDev := 0;

                               VAR_RNS_SEQ.Mem.ContainersStop := TRUE;                                                 (* STEP: 72 *)
                               VAR_RNS_SEQ.Mem.ControlInsercion := FALSE;                                              (* STEP: 72 *)
                               VAR_RNS_SEQ.Mem.ControlContinous := FALSE;                                              (* STEP: 72 *)
                               VAR_RNS_SEQ.Mem.PBAbortEnable := TRUE;                                                  (* STEP: 72 PB Abort Sequence Enable*)
                               VAR_RNS_SEQ.Mem.PBStopEnable := TRUE;                                                   (* STEP: 72 PB Stop Sequence Enable*)
                               VAR_RNS_SEQ.Mem.PBStartEnable := FALSE;                                                 (* STEP: 72 PB Start Sequence Enable*)
                               VAR_RNS_SEQ.Mem.ByPassed := FALSE;                                                      (* STEP: 72 *)
                               VAR_RNS_SEQ.Mem.InsercionDevice := TRUE;                                                (* STEP: 72 *)
                               VAR_RNS_SEQ.Mem.AirTreatmentControl := FALSE;                                           (* STEP: 72 *)
                               VAR_RNS_SEQ.Mem.WaterTreatmentControl := FALSE;                                         (* STEP: 72 *)
                               VAR_RNS_SEQ.Mem.SpeedReductionControl := TRUE;                                          (* STEP: 72 *)
                               VAR_RNS_SEQ.Mem.ByPassRequest := FALSE;                                                 (* STEP: 72 *)
                               VAR_RNS_SEQ.Mem.CopAfterCipRequest := FALSE;                                            (* STEP: 72 *)
                               VAR_RNS_SEQ.Mem.NoBoNoSprayInsercion := FALSE;                                          (* STEP: 72 *)

                               VAR_RNS_SEQ.ITC.WTT_ProductRequest := FALSE;                                            (* STEP: 72 *)
                               VAR_RNS_SEQ.ITC.WTT_ProductionRunning := FALSE;                                         (* STEP: 72 *)

                       73: (* CONTROL - Insercion Air *)

                               VAR_RNS_SEQ.Device.AVB224.AutoCnd := FALSE;                                             (* STEP: 73 AVB224*)
                               VAR_RNS_SEQ.Device.AVB224.EnableCnd := FALSE;
                               VAR_RNS_SEQ.Device.AVB228.AutoCnd := FALSE;                                             (* STEP: 73 AVB228*)
                               VAR_RNS_SEQ.Device.AVB228.EnableCnd := FALSE;
                               VAR_RNS_SEQ.Device.AVB234.AutoCnd := FALSE;                                             (* STEP: 73 AVB234*)
                               VAR_RNS_SEQ.Device.AVB234.EnableCnd := FALSE;
                               VAR_RNS_SEQ.Device.AVB261.AutoCnd := FALSE;                                             (* STEP: 73 AVB261*)
                               VAR_RNS_SEQ.Device.AVB261.EnableCnd := FALSE;
                               VAR_RNS_SEQ.Device.AVB264.AutoCnd := FALSE;                                             (* STEP: 73 AVB264*)
                               VAR_RNS_SEQ.Device.AVB264.EnableCnd := FALSE;
                               VAR_RNS_SEQ.Device.AVB265.AutoCnd := FALSE;                                             (* STEP: 73 AVB265*)
                               VAR_RNS_SEQ.Device.AVB265.EnableCnd := FALSE;
                               VAR_RNS_SEQ.Device.AVB266.AutoCnd := FALSE;                                             (* STEP: 73 AVB266*)
                               VAR_RNS_SEQ.Device.AVB266.EnableCnd := FALSE;
                               VAR_RNS_SEQ.Device.AVB267.AutoCnd := FALSE;                                             (* STEP: 73 AVB267*)
                               VAR_RNS_SEQ.Device.AVB267.EnableCnd := FALSE;
                               VAR_RNS_SEQ.Device.AVB268.AutoCnd := FALSE;                                             (* STEP: 73 AVB268*)
                               VAR_RNS_SEQ.Device.AVB268.EnableCnd := FALSE;
                               VAR_RNS_SEQ.Device.AVB273.AutoCnd := TRUE;                                              (* STEP: 73 AVB273*)
                               VAR_RNS_SEQ.Device.AVB273.EnableCnd := FALSE;
                               VAR_RNS_SEQ.Device.AVB294.AutoCnd := FALSE;                                             (* STEP: 73 AVB294*)
                               VAR_RNS_SEQ.Device.AVB294.EnableCnd := FALSE;

                               VAR_RNS_SEQ.Device.PPB209_PID.PID_Enable := FALSE;                                      (* STEP: 73 PPB209*)
                               VAR_RNS_SEQ.Device.PPB209_PID.PID_Mode := FALSE;
                               VAR_RNS_SEQ.Device.PPB209_PID.Auto_SP_Value := 0;
                               VAR_RNS_SEQ.Device.PPB209_PID.FIX_Value := 0;

                               VAR_RNS_SEQ.Device.RVB202_PID.PID_Enable := FALSE;                                      (* STEP: 73 *)
                               VAR_RNS_SEQ.Device.RVB202_PID.PID_Mode := FALSE;
                               VAR_RNS_SEQ.Device.RVB202_PID.Auto_SP_Value := 0;
                               VAR_RNS_SEQ.Device.RVB202_PID.FIX_Value := 0;

                               VAR_RNS_SEQ.Device.FSB220.ALR := FALSE;                                                 (* STEP: 73 FSB220*)
                               VAR_RNS_SEQ.Device.FSB220.WAIT_OFF := FALSE;
                               VAR_RNS_SEQ.Device.FSB220.WAIT_ON := FALSE;

                               VAR_RNS_SEQ.Device.LSB209.ALR := FALSE;                                                 (* STEP: 73 LSB209*)
                               VAR_RNS_SEQ.Device.LSB209.WAIT_OFF := FALSE;
                               VAR_RNS_SEQ.Device.LSB209.WAIT_ON := FALSE;

                               VAR_RNS_SEQ.Device.LSB210.ALR := FALSE;                                                 (* STEP: 73 LSB210*)
                               VAR_RNS_SEQ.Device.LSB210.WAIT_OFF := FALSE;
                               VAR_RNS_SEQ.Device.LSB210.WAIT_ON := FALSE;

                               VAR_RNS_SEQ.Device.LSB299.ALR := FALSE;                                                 (* STEP: 73 *)
                               VAR_RNS_SEQ.Device.LSB299.WAIT_OFF := FALSE;
                               VAR_RNS_SEQ.Device.LSB299.WAIT_ON := FALSE;

                               VAR_RNS_SEQ.Device.FSB201.ALR := FALSE;                                                 (* STEP: 73 FSB201*)
                               VAR_RNS_SEQ.Device.FSB201.WAIT_OFF := FALSE;
                               VAR_RNS_SEQ.Device.FSB201.WAIT_ON := FALSE;

                               VAR_RNS_SEQ.Device.FTB201.ALR_HighLimitEn := FALSE;                                     (* STEP: 73 FTB201*)
                               VAR_RNS_SEQ.Device.FTB201.ALR_HighLimitSP := 0;
                               VAR_RNS_SEQ.Device.FTB201.ALR_LowLimitEn := TRUE;
                               VAR_RNS_SEQ.Device.FTB201.ALR_LowLimitSP := HMI_PAR_1._166;
                               VAR_RNS_SEQ.Device.FTB201.SP := HMI_PAR_1._164;
                               VAR_RNS_SEQ.Device.FTB201.CMP := 3;
                               VAR_RNS_SEQ.Device.FTB201.MinDev := HMI_PAR_1._165;
                               VAR_RNS_SEQ.Device.FTB201.MaxDev := 2*HMI_PAR_1._165;

                               VAR_RNS_SEQ.Device.FTB202.ALR_HighLimitEn := FALSE;                                     (* STEP: 73 FTB202*)
                               VAR_RNS_SEQ.Device.FTB202.ALR_HighLimitSP := 0;
                               VAR_RNS_SEQ.Device.FTB202.ALR_LowLimitEn := FALSE;
                               VAR_RNS_SEQ.Device.FTB202.ALR_LowLimitSP := 0;
                               VAR_RNS_SEQ.Device.FTB202.SP := 0;
                               VAR_RNS_SEQ.Device.FTB202.CMP := 0;
                               VAR_RNS_SEQ.Device.FTB202.MinDev := 0;
                               VAR_RNS_SEQ.Device.FTB202.MaxDev := 0;

                               VAR_RNS_SEQ.Device.PTB220.ALR_HighLimitEn := FALSE;                                     (* STEP: 73 PTB220*)
                               VAR_RNS_SEQ.Device.PTB220.ALR_HighLimitSP := 0;
                               VAR_RNS_SEQ.Device.PTB220.ALR_LowLimitEn := FALSE;
                               VAR_RNS_SEQ.Device.PTB220.ALR_LowLimitSP := 0;
                               VAR_RNS_SEQ.Device.PTB220.SP := 0;
                               VAR_RNS_SEQ.Device.PTB220.CMP := 0;
                               VAR_RNS_SEQ.Device.PTB220.MinDev := 0;
                               VAR_RNS_SEQ.Device.PTB220.MaxDev := 0;

                               VAR_RNS_SEQ.Device.PTB270.ALR_HighLimitEn := FALSE;                                     (* STEP: 73 PTB270*)
                               VAR_RNS_SEQ.Device.PTB270.ALR_HighLimitSP := 0;
                               VAR_RNS_SEQ.Device.PTB270.ALR_LowLimitEn := FALSE;
                               VAR_RNS_SEQ.Device.PTB270.ALR_LowLimitSP := 0;
                               VAR_RNS_SEQ.Device.PTB270.SP := 0;
                               VAR_RNS_SEQ.Device.PTB270.CMP := 0;
                               VAR_RNS_SEQ.Device.PTB270.MinDev := 0;
                               VAR_RNS_SEQ.Device.PTB270.MaxDev := 0;

                               VAR_RNS_SEQ.Device.LTB202.ALR_HighLimitEn := FALSE;                                     (* STEP: 73 LTB202*)
                               VAR_RNS_SEQ.Device.LTB202.ALR_HighLimitSP := 0;
                               VAR_RNS_SEQ.Device.LTB202.ALR_LowLimitEn := FALSE;
                               VAR_RNS_SEQ.Device.LTB202.ALR_LowLimitSP := 0;
                               VAR_RNS_SEQ.Device.LTB202.SP := 0;
                               VAR_RNS_SEQ.Device.LTB202.CMP := 0;
                               VAR_RNS_SEQ.Device.LTB202.MinDev := 0;
                               VAR_RNS_SEQ.Device.LTB202.MaxDev := 0;

                               VAR_RNS_SEQ.Device.PTB290.ALR_HighLimitEn := FALSE;                                     (* STEP: 73 PTB290*)
                               VAR_RNS_SEQ.Device.PTB290.ALR_HighLimitSP := 0;
                               VAR_RNS_SEQ.Device.PTB290.ALR_LowLimitEn := FALSE;
                               VAR_RNS_SEQ.Device.PTB290.ALR_LowLimitSP := 0;
                               VAR_RNS_SEQ.Device.PTB290.SP := 0;
                               VAR_RNS_SEQ.Device.PTB290.CMP := 0;
                               VAR_RNS_SEQ.Device.PTB290.MinDev := 0;
                               VAR_RNS_SEQ.Device.PTB290.MaxDev := 0;

                               VAR_RNS_SEQ.Mem.ContainersStop := TRUE;                                                 (* STEP: 73 *)
                               VAR_RNS_SEQ.Mem.ControlInsercion := TRUE;                                               (* STEP: 73 *)
                               VAR_RNS_SEQ.Mem.ControlContinous := FALSE;                                              (* STEP: 73 *)
                               VAR_RNS_SEQ.Mem.PBAbortEnable := TRUE;                                                  (* STEP: 73 PB Abort Sequence Enable*)
                               VAR_RNS_SEQ.Mem.PBStopEnable := TRUE;                                                   (* STEP: 73 PB Stop Sequence Enable*)
                               VAR_RNS_SEQ.Mem.PBStartEnable := FALSE;                                                 (* STEP: 73 PB Start Sequence Enable*)
                               VAR_RNS_SEQ.Mem.ByPassed := FALSE;                                                      (* STEP: 73 *)
                               VAR_RNS_SEQ.Mem.InsercionDevice := TRUE;                                                (* STEP: 73 *)
                               VAR_RNS_SEQ.Mem.AirTreatmentControl := TRUE;                                            (* STEP: 73 *)
                               VAR_RNS_SEQ.Mem.WaterTreatmentControl := FALSE;                                         (* STEP: 73 *)
                               VAR_RNS_SEQ.Mem.SpeedReductionControl := TRUE;                                          (* STEP: 73 *)
                               VAR_RNS_SEQ.Mem.ByPassRequest := FALSE;                                                 (* STEP: 73 *)
                               VAR_RNS_SEQ.Mem.CopAfterCipRequest := FALSE;                                            (* STEP: 73 *)
                               VAR_RNS_SEQ.Mem.NoBoNoSprayInsercion := FALSE;                                          (* STEP: 73 *)

                               VAR_RNS_SEQ.ITC.WTT_ProductRequest := FALSE;                                            (* STEP: 73 *)
                               VAR_RNS_SEQ.ITC.WTT_ProductionRunning := FALSE;                                         (* STEP: 73 *)

                       74: (* CONTROL - Water Startup I *)

                               VAR_RNS_SEQ.Device.AVB224.AutoCnd := FALSE;                                             (* STEP: 74 AVB224*)
                               VAR_RNS_SEQ.Device.AVB224.EnableCnd := FALSE;
                               VAR_RNS_SEQ.Device.AVB228.AutoCnd := FALSE;                                             (* STEP: 74 AVB228*)
                               VAR_RNS_SEQ.Device.AVB228.EnableCnd := FALSE;
                               VAR_RNS_SEQ.Device.AVB234.AutoCnd := FALSE;                                             (* STEP: 74 AVB234*)
                               VAR_RNS_SEQ.Device.AVB234.EnableCnd := FALSE;
                               VAR_RNS_SEQ.Device.AVB261.AutoCnd := TRUE;                                              (* STEP: 74 AVB261*)
                               VAR_RNS_SEQ.Device.AVB261.EnableCnd := FALSE;
                               VAR_RNS_SEQ.Device.AVB264.AutoCnd := TRUE;                                              (* STEP: 74 AVB264*)
                               VAR_RNS_SEQ.Device.AVB264.EnableCnd := FALSE;
                               VAR_RNS_SEQ.Device.AVB265.AutoCnd := TRUE;                                              (* STEP: 74 AVB265*)
                               VAR_RNS_SEQ.Device.AVB265.EnableCnd := FALSE;
                               VAR_RNS_SEQ.Device.AVB266.AutoCnd := FALSE;                                             (* STEP: 74 AVB266*)
                               VAR_RNS_SEQ.Device.AVB266.EnableCnd := FALSE;
                               VAR_RNS_SEQ.Device.AVB267.AutoCnd := FALSE;                                             (* STEP: 74 AVB267*)
                               VAR_RNS_SEQ.Device.AVB267.EnableCnd := FALSE;
                               VAR_RNS_SEQ.Device.AVB268.AutoCnd := FALSE;                                             (* STEP: 74 AVB268*)
                               VAR_RNS_SEQ.Device.AVB268.EnableCnd := FALSE;
                               VAR_RNS_SEQ.Device.AVB273.AutoCnd := FALSE;                                             (* STEP: 74 AVB273*)
                               VAR_RNS_SEQ.Device.AVB273.EnableCnd := FALSE;
                               VAR_RNS_SEQ.Device.AVB294.AutoCnd := FALSE;                                             (* STEP: 74 AVB294*)
                               VAR_RNS_SEQ.Device.AVB294.EnableCnd := FALSE;

                               VAR_RNS_SEQ.Device.PPB209_PID.PID_Enable := FALSE;                                      (* STEP: 74 PPB209*)
                               VAR_RNS_SEQ.Device.PPB209_PID.PID_Mode := FALSE;
                               VAR_RNS_SEQ.Device.PPB209_PID.Auto_SP_Value := 0;
                               VAR_RNS_SEQ.Device.PPB209_PID.FIX_Value := 0;

                               VAR_RNS_SEQ.Device.RVB202_PID.PID_Enable := TRUE;                                       (* STEP: 74 *)
                               VAR_RNS_SEQ.Device.RVB202_PID.PID_Mode := FALSE;
                               VAR_RNS_SEQ.Device.RVB202_PID.Auto_SP_Value := 0;
                               VAR_RNS_SEQ.Device.RVB202_PID.FIX_Value := HMI_PAM_1._092;

                               VAR_RNS_SEQ.Device.FSB220.ALR := TRUE;                                                  (* STEP: 74 FSB220*)
                               VAR_RNS_SEQ.Device.FSB220.WAIT_OFF := FALSE;
                               VAR_RNS_SEQ.Device.FSB220.WAIT_ON := TRUE;

                               VAR_RNS_SEQ.Device.LSB209.ALR := FALSE;                                                 (* STEP: 74 LSB209*)
                               VAR_RNS_SEQ.Device.LSB209.WAIT_OFF := FALSE;
                               VAR_RNS_SEQ.Device.LSB209.WAIT_ON := FALSE;

                               VAR_RNS_SEQ.Device.LSB210.ALR := FALSE;                                                 (* STEP: 74 LSB210*)
                               VAR_RNS_SEQ.Device.LSB210.WAIT_OFF := FALSE;
                               VAR_RNS_SEQ.Device.LSB210.WAIT_ON := FALSE;

                               VAR_RNS_SEQ.Device.LSB299.ALR := FALSE;                                                 (* STEP: 74 *)
                               VAR_RNS_SEQ.Device.LSB299.WAIT_OFF := FALSE;
                               VAR_RNS_SEQ.Device.LSB299.WAIT_ON := FALSE;

                               VAR_RNS_SEQ.Device.FSB201.ALR := FALSE;                                                 (* STEP: 74 FSB201*)
                               VAR_RNS_SEQ.Device.FSB201.WAIT_OFF := FALSE;
                               VAR_RNS_SEQ.Device.FSB201.WAIT_ON := FALSE;

                               VAR_RNS_SEQ.Device.FTB201.ALR_HighLimitEn := FALSE;                                     (* STEP: 74 FTB201*)
                               VAR_RNS_SEQ.Device.FTB201.ALR_HighLimitSP := 0;
                               VAR_RNS_SEQ.Device.FTB201.ALR_LowLimitEn := FALSE;
                               VAR_RNS_SEQ.Device.FTB201.ALR_LowLimitSP := 0;
                               VAR_RNS_SEQ.Device.FTB201.SP := 0;
                               VAR_RNS_SEQ.Device.FTB201.CMP := 0;
                               VAR_RNS_SEQ.Device.FTB201.MinDev := 0;
                               VAR_RNS_SEQ.Device.FTB201.MaxDev := 0;

                               VAR_RNS_SEQ.Device.FTB202.ALR_HighLimitEn := FALSE;                                     (* STEP: 74 FTB202*)
                               VAR_RNS_SEQ.Device.FTB202.ALR_HighLimitSP := 0;
                               VAR_RNS_SEQ.Device.FTB202.ALR_LowLimitEn := TRUE;
                               VAR_RNS_SEQ.Device.FTB202.ALR_LowLimitSP := HMI_PAR_1._169;
                               VAR_RNS_SEQ.Device.FTB202.SP := HMI_PAR_1._167;
                               VAR_RNS_SEQ.Device.FTB202.CMP := 3;
                               VAR_RNS_SEQ.Device.FTB202.MinDev := HMI_PAR_1._168;
                               VAR_RNS_SEQ.Device.FTB202.MaxDev := HMI_PAR_1._168 * 2;

                               VAR_RNS_SEQ.Device.PTB220.ALR_HighLimitEn := FALSE;                                     (* STEP: 74 PTB220*)
                               VAR_RNS_SEQ.Device.PTB220.ALR_HighLimitSP := 0;
                               VAR_RNS_SEQ.Device.PTB220.ALR_LowLimitEn := TRUE;
                               VAR_RNS_SEQ.Device.PTB220.ALR_LowLimitSP := HMI_PAM_1._092     *0.80;
                               VAR_RNS_SEQ.Device.PTB220.SP := HMI_PAM_1._092;
                               VAR_RNS_SEQ.Device.PTB220.CMP := 2;
                               VAR_RNS_SEQ.Device.PTB220.MinDev := 0;
                               VAR_RNS_SEQ.Device.PTB220.MaxDev := 0;

                               VAR_RNS_SEQ.Device.PTB270.ALR_HighLimitEn := FALSE;                                     (* STEP: 74 PTB270*)
                               VAR_RNS_SEQ.Device.PTB270.ALR_HighLimitSP := 0;
                               VAR_RNS_SEQ.Device.PTB270.ALR_LowLimitEn := FALSE;
                               VAR_RNS_SEQ.Device.PTB270.ALR_LowLimitSP := 0;
                               VAR_RNS_SEQ.Device.PTB270.SP := 0;
                               VAR_RNS_SEQ.Device.PTB270.CMP := 0;
                               VAR_RNS_SEQ.Device.PTB270.MinDev := 0;
                               VAR_RNS_SEQ.Device.PTB270.MaxDev := 0;

                               VAR_RNS_SEQ.Device.LTB202.ALR_HighLimitEn := FALSE;                                     (* STEP: 74 LTB202*)
                               VAR_RNS_SEQ.Device.LTB202.ALR_HighLimitSP := 0;
                               VAR_RNS_SEQ.Device.LTB202.ALR_LowLimitEn := FALSE;
                               VAR_RNS_SEQ.Device.LTB202.ALR_LowLimitSP := 0;
                               VAR_RNS_SEQ.Device.LTB202.SP := 0;
                               VAR_RNS_SEQ.Device.LTB202.CMP := 0;
                               VAR_RNS_SEQ.Device.LTB202.MinDev := 0;
                               VAR_RNS_SEQ.Device.LTB202.MaxDev := 0;

                               VAR_RNS_SEQ.Device.PTB290.ALR_HighLimitEn := FALSE;                                     (* STEP: 74 PTB290*)
                               VAR_RNS_SEQ.Device.PTB290.ALR_HighLimitSP := 0;
                               VAR_RNS_SEQ.Device.PTB290.ALR_LowLimitEn := FALSE;
                               VAR_RNS_SEQ.Device.PTB290.ALR_LowLimitSP := 0;
                               VAR_RNS_SEQ.Device.PTB290.SP := 0;
                               VAR_RNS_SEQ.Device.PTB290.CMP := 0;
                               VAR_RNS_SEQ.Device.PTB290.MinDev := 0;
                               VAR_RNS_SEQ.Device.PTB290.MaxDev := 0;

                               VAR_RNS_SEQ.Mem.ContainersStop := TRUE;                                                 (* STEP: 74 *)
                               VAR_RNS_SEQ.Mem.ControlInsercion := FALSE;                                              (* STEP: 74 *)
                               VAR_RNS_SEQ.Mem.ControlContinous := FALSE;                                              (* STEP: 74 *)
                               VAR_RNS_SEQ.Mem.PBAbortEnable := TRUE;                                                  (* STEP: 74 PB Abort Sequence Enable*)
                               VAR_RNS_SEQ.Mem.PBStopEnable := TRUE;                                                   (* STEP: 74 PB Stop Sequence Enable*)
                               VAR_RNS_SEQ.Mem.PBStartEnable := FALSE;                                                 (* STEP: 74 PB Start Sequence Enable*)
                               VAR_RNS_SEQ.Mem.ByPassed := FALSE;                                                      (* STEP: 74 *)
                               VAR_RNS_SEQ.Mem.InsercionDevice := TRUE;                                                (* STEP: 74 *)
                               VAR_RNS_SEQ.Mem.AirTreatmentControl := FALSE;                                           (* STEP: 74 *)
                               VAR_RNS_SEQ.Mem.WaterTreatmentControl := FALSE;                                         (* STEP: 74 *)
                               VAR_RNS_SEQ.Mem.SpeedReductionControl := TRUE;                                          (* STEP: 74 *)
                               VAR_RNS_SEQ.Mem.ByPassRequest := FALSE;                                                 (* STEP: 74 *)
                               VAR_RNS_SEQ.Mem.CopAfterCipRequest := FALSE;                                            (* STEP: 74 *)
                               VAR_RNS_SEQ.Mem.NoBoNoSprayInsercion := TRUE;                                           (* STEP: 74 *)

                               VAR_RNS_SEQ.ITC.WTT_ProductRequest := TRUE;                                             (* STEP: 74 *)
                               VAR_RNS_SEQ.ITC.WTT_ProductionRunning := FALSE;                                         (* STEP: 74 *)

                       75: (* CONTROL - Insercion Water *)

                               VAR_RNS_SEQ.Device.AVB224.AutoCnd := FALSE;                                             (* STEP: 75 AVB224*)
                               VAR_RNS_SEQ.Device.AVB224.EnableCnd := FALSE;
                               VAR_RNS_SEQ.Device.AVB228.AutoCnd := FALSE;                                             (* STEP: 75 AVB228*)
                               VAR_RNS_SEQ.Device.AVB228.EnableCnd := FALSE;
                               VAR_RNS_SEQ.Device.AVB234.AutoCnd := FALSE;                                             (* STEP: 75 AVB234*)
                               VAR_RNS_SEQ.Device.AVB234.EnableCnd := FALSE;
                               VAR_RNS_SEQ.Device.AVB261.AutoCnd := TRUE;                                              (* STEP: 75 AVB261*)
                               VAR_RNS_SEQ.Device.AVB261.EnableCnd := FALSE;
                               VAR_RNS_SEQ.Device.AVB264.AutoCnd := TRUE;                                              (* STEP: 75 AVB264*)
                               VAR_RNS_SEQ.Device.AVB264.EnableCnd := FALSE;
                               VAR_RNS_SEQ.Device.AVB265.AutoCnd := TRUE;                                              (* STEP: 75 AVB265*)
                               VAR_RNS_SEQ.Device.AVB265.EnableCnd := FALSE;
                               VAR_RNS_SEQ.Device.AVB266.AutoCnd := FALSE;                                             (* STEP: 75 AVB266*)
                               VAR_RNS_SEQ.Device.AVB266.EnableCnd := FALSE;
                               VAR_RNS_SEQ.Device.AVB267.AutoCnd := FALSE;                                             (* STEP: 75 AVB267*)
                               VAR_RNS_SEQ.Device.AVB267.EnableCnd := FALSE;
                               VAR_RNS_SEQ.Device.AVB268.AutoCnd := FALSE;                                             (* STEP: 75 AVB268*)
                               VAR_RNS_SEQ.Device.AVB268.EnableCnd := FALSE;
                               VAR_RNS_SEQ.Device.AVB273.AutoCnd := FALSE;                                             (* STEP: 75 AVB273*)
                               VAR_RNS_SEQ.Device.AVB273.EnableCnd := FALSE;
                               VAR_RNS_SEQ.Device.AVB294.AutoCnd := FALSE;                                             (* STEP: 75 AVB294*)
                               VAR_RNS_SEQ.Device.AVB294.EnableCnd := FALSE;

                               VAR_RNS_SEQ.Device.PPB209_PID.PID_Enable := FALSE;                                      (* STEP: 75 PPB209*)
                               VAR_RNS_SEQ.Device.PPB209_PID.PID_Mode := FALSE;
                               VAR_RNS_SEQ.Device.PPB209_PID.Auto_SP_Value := 0;
                               VAR_RNS_SEQ.Device.PPB209_PID.FIX_Value := 0;

                               VAR_RNS_SEQ.Device.RVB202_PID.PID_Enable := TRUE;                                       (* STEP: 75 *)
                               VAR_RNS_SEQ.Device.RVB202_PID.PID_Mode := FALSE;
                               VAR_RNS_SEQ.Device.RVB202_PID.Auto_SP_Value := 0;
                               VAR_RNS_SEQ.Device.RVB202_PID.FIX_Value := HMI_PAM_1._092;

                               VAR_RNS_SEQ.Device.FSB220.ALR := FALSE;                                                 (* STEP: 75 FSB220*)
                               VAR_RNS_SEQ.Device.FSB220.WAIT_OFF := FALSE;
                               VAR_RNS_SEQ.Device.FSB220.WAIT_ON := FALSE;

                               VAR_RNS_SEQ.Device.LSB209.ALR := FALSE;                                                 (* STEP: 75 LSB209*)
                               VAR_RNS_SEQ.Device.LSB209.WAIT_OFF := FALSE;
                               VAR_RNS_SEQ.Device.LSB209.WAIT_ON := FALSE;

                               VAR_RNS_SEQ.Device.LSB210.ALR := FALSE;                                                 (* STEP: 75 LSB210*)
                               VAR_RNS_SEQ.Device.LSB210.WAIT_OFF := FALSE;
                               VAR_RNS_SEQ.Device.LSB210.WAIT_ON := FALSE;

                               VAR_RNS_SEQ.Device.LSB299.ALR := FALSE;                                                 (* STEP: 75 *)
                               VAR_RNS_SEQ.Device.LSB299.WAIT_OFF := FALSE;
                               VAR_RNS_SEQ.Device.LSB299.WAIT_ON := FALSE;

                               VAR_RNS_SEQ.Device.FSB201.ALR := FALSE;                                                 (* STEP: 75 FSB201*)
                               VAR_RNS_SEQ.Device.FSB201.WAIT_OFF := FALSE;
                               VAR_RNS_SEQ.Device.FSB201.WAIT_ON := FALSE;

                               VAR_RNS_SEQ.Device.FTB201.ALR_HighLimitEn := FALSE;                                     (* STEP: 75 FTB201*)
                               VAR_RNS_SEQ.Device.FTB201.ALR_HighLimitSP := 0;
                               VAR_RNS_SEQ.Device.FTB201.ALR_LowLimitEn := FALSE;
                               VAR_RNS_SEQ.Device.FTB201.ALR_LowLimitSP := 0;
                               VAR_RNS_SEQ.Device.FTB201.SP := 0;
                               VAR_RNS_SEQ.Device.FTB201.CMP := 0;
                               VAR_RNS_SEQ.Device.FTB201.MinDev := 0;
                               VAR_RNS_SEQ.Device.FTB201.MaxDev := 0;

                               VAR_RNS_SEQ.Device.FTB202.ALR_HighLimitEn := FALSE;                                     (* STEP: 75 FTB202*)
                               VAR_RNS_SEQ.Device.FTB202.ALR_HighLimitSP := 0;
                               VAR_RNS_SEQ.Device.FTB202.ALR_LowLimitEn := TRUE;
                               VAR_RNS_SEQ.Device.FTB202.ALR_LowLimitSP := HMI_PAR_1._169;
                               VAR_RNS_SEQ.Device.FTB202.SP := HMI_PAR_1._167;
                               VAR_RNS_SEQ.Device.FTB202.CMP := 3;
                               VAR_RNS_SEQ.Device.FTB202.MinDev := HMI_PAR_1._168;
                               VAR_RNS_SEQ.Device.FTB202.MaxDev := HMI_PAR_1._168 * 2;

                               VAR_RNS_SEQ.Device.PTB220.ALR_HighLimitEn := FALSE;                                     (* STEP: 75 PTB220*)
                               VAR_RNS_SEQ.Device.PTB220.ALR_HighLimitSP := 0;
                               VAR_RNS_SEQ.Device.PTB220.ALR_LowLimitEn := TRUE;
                               VAR_RNS_SEQ.Device.PTB220.ALR_LowLimitSP := HMI_PAM_1._092     *0.80;
                               VAR_RNS_SEQ.Device.PTB220.SP := HMI_PAM_1._092;
                               VAR_RNS_SEQ.Device.PTB220.CMP := 2;
                               VAR_RNS_SEQ.Device.PTB220.MinDev := 0;
                               VAR_RNS_SEQ.Device.PTB220.MaxDev := 0;

                               VAR_RNS_SEQ.Device.PTB270.ALR_HighLimitEn := FALSE;                                     (* STEP: 75 PTB270*)
                               VAR_RNS_SEQ.Device.PTB270.ALR_HighLimitSP := 0;
                               VAR_RNS_SEQ.Device.PTB270.ALR_LowLimitEn := FALSE;
                               VAR_RNS_SEQ.Device.PTB270.ALR_LowLimitSP := 0;
                               VAR_RNS_SEQ.Device.PTB270.SP := 0;
                               VAR_RNS_SEQ.Device.PTB270.CMP := 0;
                               VAR_RNS_SEQ.Device.PTB270.MinDev := 0;
                               VAR_RNS_SEQ.Device.PTB270.MaxDev := 0;

                               VAR_RNS_SEQ.Device.LTB202.ALR_HighLimitEn := FALSE;                                     (* STEP: 75 LTB202*)
                               VAR_RNS_SEQ.Device.LTB202.ALR_HighLimitSP := 0;
                               VAR_RNS_SEQ.Device.LTB202.ALR_LowLimitEn := FALSE;
                               VAR_RNS_SEQ.Device.LTB202.ALR_LowLimitSP := 0;
                               VAR_RNS_SEQ.Device.LTB202.SP := 0;
                               VAR_RNS_SEQ.Device.LTB202.CMP := 0;
                               VAR_RNS_SEQ.Device.LTB202.MinDev := 0;
                               VAR_RNS_SEQ.Device.LTB202.MaxDev := 0;

                               VAR_RNS_SEQ.Device.PTB290.ALR_HighLimitEn := FALSE;                                     (* STEP: 75 PTB290*)
                               VAR_RNS_SEQ.Device.PTB290.ALR_HighLimitSP := 0;
                               VAR_RNS_SEQ.Device.PTB290.ALR_LowLimitEn := FALSE;
                               VAR_RNS_SEQ.Device.PTB290.ALR_LowLimitSP := 0;
                               VAR_RNS_SEQ.Device.PTB290.SP := 0;
                               VAR_RNS_SEQ.Device.PTB290.CMP := 0;
                               VAR_RNS_SEQ.Device.PTB290.MinDev := 0;
                               VAR_RNS_SEQ.Device.PTB290.MaxDev := 0;

                               VAR_RNS_SEQ.Mem.ContainersStop := TRUE;                                                 (* STEP: 75 *)
                               VAR_RNS_SEQ.Mem.ControlInsercion := TRUE;                                               (* STEP: 75 *)
                               VAR_RNS_SEQ.Mem.ControlContinous := FALSE;                                              (* STEP: 75 *)
                               VAR_RNS_SEQ.Mem.PBAbortEnable := TRUE;                                                  (* STEP: 75 PB Abort Sequence Enable*)
                               VAR_RNS_SEQ.Mem.PBStopEnable := TRUE;                                                   (* STEP: 75 PB Stop Sequence Enable*)
                               VAR_RNS_SEQ.Mem.PBStartEnable := FALSE;                                                 (* STEP: 75 PB Start Sequence Enable*)
                               VAR_RNS_SEQ.Mem.ByPassed := FALSE;                                                      (* STEP: 75 *)
                               VAR_RNS_SEQ.Mem.InsercionDevice := TRUE;                                                (* STEP: 75 *)
                               VAR_RNS_SEQ.Mem.AirTreatmentControl := FALSE;                                           (* STEP: 75 *)
                               VAR_RNS_SEQ.Mem.WaterTreatmentControl := TRUE;                                          (* STEP: 75 *)
                               VAR_RNS_SEQ.Mem.SpeedReductionControl := TRUE;                                          (* STEP: 75 *)
                               VAR_RNS_SEQ.Mem.ByPassRequest := FALSE;                                                 (* STEP: 75 *)
                               VAR_RNS_SEQ.Mem.CopAfterCipRequest := FALSE;                                            (* STEP: 75 *)
                               VAR_RNS_SEQ.Mem.NoBoNoSprayInsercion := TRUE;                                           (* STEP: 75 *)

                               VAR_RNS_SEQ.ITC.WTT_ProductRequest := TRUE;                                             (* STEP: 75 *)
                               VAR_RNS_SEQ.ITC.WTT_ProductionRunning := TRUE;                                          (* STEP: 75 *)

                       76: (* CONTROL - Air Startup C *)

                               VAR_RNS_SEQ.Device.AVB224.AutoCnd := TRUE;                                              (* STEP: 76 AVB224*)
                               VAR_RNS_SEQ.Device.AVB224.EnableCnd := TRUE;
                               VAR_RNS_SEQ.Device.AVB228.AutoCnd := FALSE;                                             (* STEP: 76 AVB228*)
                               VAR_RNS_SEQ.Device.AVB228.EnableCnd := FALSE;
                               VAR_RNS_SEQ.Device.AVB234.AutoCnd := FALSE;                                             (* STEP: 76 AVB234*)
                               VAR_RNS_SEQ.Device.AVB234.EnableCnd := FALSE;
                               VAR_RNS_SEQ.Device.AVB261.AutoCnd := TRUE;                                              (* STEP: 76 AVB261*)
                               VAR_RNS_SEQ.Device.AVB261.EnableCnd := TRUE;
                               VAR_RNS_SEQ.Device.AVB264.AutoCnd := TRUE;                                              (* STEP: 76 AVB264*)
                               VAR_RNS_SEQ.Device.AVB264.EnableCnd := TRUE;
                               VAR_RNS_SEQ.Device.AVB265.AutoCnd := TRUE;                                              (* STEP: 76 AVB265*)
                               VAR_RNS_SEQ.Device.AVB265.EnableCnd := TRUE;
                               VAR_RNS_SEQ.Device.AVB266.AutoCnd := FALSE;                                             (* STEP: 76 AVB266*)
                               VAR_RNS_SEQ.Device.AVB266.EnableCnd := FALSE;
                               VAR_RNS_SEQ.Device.AVB267.AutoCnd := FALSE;                                             (* STEP: 76 AVB267*)
                               VAR_RNS_SEQ.Device.AVB267.EnableCnd := FALSE;
                               VAR_RNS_SEQ.Device.AVB268.AutoCnd := FALSE;                                             (* STEP: 76 AVB268*)
                               VAR_RNS_SEQ.Device.AVB268.EnableCnd := FALSE;
                               VAR_RNS_SEQ.Device.AVB273.AutoCnd := TRUE;                                              (* STEP: 76 AVB273*)
                               VAR_RNS_SEQ.Device.AVB273.EnableCnd := FALSE;
                               VAR_RNS_SEQ.Device.AVB294.AutoCnd := FALSE;                                             (* STEP: 76 AVB294*)
                               VAR_RNS_SEQ.Device.AVB294.EnableCnd := FALSE;

                               VAR_RNS_SEQ.Device.PPB209_PID.PID_Enable := FALSE;                                      (* STEP: 76 PPB209*)
                               VAR_RNS_SEQ.Device.PPB209_PID.PID_Mode := FALSE;
                               VAR_RNS_SEQ.Device.PPB209_PID.Auto_SP_Value := 0;
                               VAR_RNS_SEQ.Device.PPB209_PID.FIX_Value := 0;

                               VAR_RNS_SEQ.Device.RVB202_PID.PID_Enable := FALSE;                                      (* STEP: 76 *)
                               VAR_RNS_SEQ.Device.RVB202_PID.PID_Mode := FALSE;
                               VAR_RNS_SEQ.Device.RVB202_PID.Auto_SP_Value := 0;
                               VAR_RNS_SEQ.Device.RVB202_PID.FIX_Value := 0;

                               VAR_RNS_SEQ.Device.FSB220.ALR := FALSE;                                                 (* STEP: 76 FSB220*)
                               VAR_RNS_SEQ.Device.FSB220.WAIT_OFF := FALSE;
                               VAR_RNS_SEQ.Device.FSB220.WAIT_ON := FALSE;

                               VAR_RNS_SEQ.Device.LSB209.ALR := FALSE;                                                 (* STEP: 76 LSB209*)
                               VAR_RNS_SEQ.Device.LSB209.WAIT_OFF := FALSE;
                               VAR_RNS_SEQ.Device.LSB209.WAIT_ON := FALSE;

                               VAR_RNS_SEQ.Device.LSB210.ALR := FALSE;                                                 (* STEP: 76 LSB210*)
                               VAR_RNS_SEQ.Device.LSB210.WAIT_OFF := FALSE;
                               VAR_RNS_SEQ.Device.LSB210.WAIT_ON := FALSE;

                               VAR_RNS_SEQ.Device.LSB299.ALR := FALSE;                                                 (* STEP: 76 *)
                               VAR_RNS_SEQ.Device.LSB299.WAIT_OFF := FALSE;
                               VAR_RNS_SEQ.Device.LSB299.WAIT_ON := FALSE;

                               VAR_RNS_SEQ.Device.FSB201.ALR := FALSE;                                                 (* STEP: 76 FSB201*)
                               VAR_RNS_SEQ.Device.FSB201.WAIT_OFF := FALSE;
                               VAR_RNS_SEQ.Device.FSB201.WAIT_ON := FALSE;

                               VAR_RNS_SEQ.Device.FTB201.ALR_HighLimitEn := FALSE;                                     (* STEP: 76 FTB201*)
                               VAR_RNS_SEQ.Device.FTB201.ALR_HighLimitSP := 0;
                               VAR_RNS_SEQ.Device.FTB201.ALR_LowLimitEn := TRUE;
                               VAR_RNS_SEQ.Device.FTB201.ALR_LowLimitSP := HMI_PAR_1._166;
                               VAR_RNS_SEQ.Device.FTB201.SP := HMI_PAR_1._164;
                               VAR_RNS_SEQ.Device.FTB201.CMP := 3;
                               VAR_RNS_SEQ.Device.FTB201.MinDev := HMI_PAR_1._165;
                               VAR_RNS_SEQ.Device.FTB201.MaxDev := 2*HMI_PAR_1._165;

                               VAR_RNS_SEQ.Device.FTB202.ALR_HighLimitEn := FALSE;                                     (* STEP: 76 FTB202*)
                               VAR_RNS_SEQ.Device.FTB202.ALR_HighLimitSP := 0;
                               VAR_RNS_SEQ.Device.FTB202.ALR_LowLimitEn := FALSE;
                               VAR_RNS_SEQ.Device.FTB202.ALR_LowLimitSP := 0;
                               VAR_RNS_SEQ.Device.FTB202.SP := 0;
                               VAR_RNS_SEQ.Device.FTB202.CMP := 0;
                               VAR_RNS_SEQ.Device.FTB202.MinDev := 0;
                               VAR_RNS_SEQ.Device.FTB202.MaxDev := 0;

                               VAR_RNS_SEQ.Device.PTB220.ALR_HighLimitEn := FALSE;                                     (* STEP: 76 PTB220*)
                               VAR_RNS_SEQ.Device.PTB220.ALR_HighLimitSP := 0;
                               VAR_RNS_SEQ.Device.PTB220.ALR_LowLimitEn := FALSE;
                               VAR_RNS_SEQ.Device.PTB220.ALR_LowLimitSP := 0;
                               VAR_RNS_SEQ.Device.PTB220.SP := 0;
                               VAR_RNS_SEQ.Device.PTB220.CMP := 0;
                               VAR_RNS_SEQ.Device.PTB220.MinDev := 0;
                               VAR_RNS_SEQ.Device.PTB220.MaxDev := 0;
```
